FUNCTION F_COEF_AR : REAL
VAR_INPUT
END_VAR
VAR

END_VAR

END_FUNCTION

(* stored: Version 1.1.0.1, ProductVersion 3.1.4022.18
   POU F_COEF_AR: Id {2f1670b1-1c15-440a-a716-93f242c11d81}, SpecialFunc None *)
